(*
Nazwa:			P13_BottleTransfer
Opis:			Stacja odkładania butelek w różne miejsca
Wersja:			v0.1
Data:			2018-10-10
Autor:			DP
Urzadzenia:		
Konfiguracja:	
Info:

*)
PROGRAM P13_BottleTransfer
VAR_INPUT
	IbFirstFormCheckFormSensor				AT %I*	: BOOL; 						// Sygnal pierwszej formatki
	IbSecondFormCheckFormSensor				AT %I*	: BOOL; 						// Sygnal drugiej formatki
	IbBottleCheckAfterBottleTransferSensor	AT %I*	: BOOL; 						// Wejście z czujnika wykrycia butelki za robotem
	IbBottleTransferFormAfterSensor			AT %I*: BOOL; 					// Czujnik formatki za robotem
	IbBottleTransferFormAfterSensor2			AT %I*: BOOL; 					// Czujnik 2 formatki za robotem
END_VAR
VAR
	// Blok Sterujący podajnikiem nakrętek
	fbBottleTransfer									: FB_Robot2Bottles;
	tonEnableDelay: TON;
	eBottleTransferState					: E_Station;
	eBottleTransferRunningState				: E_RobotMovState;	
	fbBottleTransferState					: FB_State;	
	
	// WEJSCIA I WYJSCIA SPRZETOWE	
	QaDataRobotIO                            AT %Q*: ARRAY[1..8] OF USINT;
    QaDataRobotREG                           AT %Q*: ARRAY[1..32] OF UINT;
    IaDataRobotIO                            AT %I*: ARRAY[1..8] OF USINT;
    IaDataRobotREG                       	 AT %I*: ARRAY[1..32] OF UINT;
	

	
	
	TimerBottleTransferEnable: TOF;
	(*Nowe od robota Mitsubishi*)
	QbBottleTransferRobotMode1 AT %Q*:BOOL; 								//Zezwalanie na pracę robota 1
	QbBottleTransferRobotMode2 AT %Q*:BOOL; 								//Zezwalanie na pracę robota 2	

//	
	
	bBottleTransferLubricationResetCase: INT;
	tonBottleTransferLubricationResetCase1: TON;
	tonBottleTransferLubricationResetCase2: TON;
	tonBottleTransferLubricationResetCase3: TON;
	tonBottleTransferLubricationResetCase4: TON;
	tonBottleTransferLubricationResetCase5: TON;
	tonBottleTransferLubricationResetCase6: TON;
	tonBottleTransferLubricationResetCase7: TON;
	bTestWarning							: BOOL;
	bTestHoming								: BOOL;
	bTestPick								: BOOL;
	bTestPlace								: BOOL;
END_VAR

IF VIS.iBottleTransferPickOffsetZShow > 40	THEN
	VIS.iBottleTransferPickOffsetZShow								:= 40;
END_IF
IF VIS.iBottleTransferPickOffsetZShow < -60	THEN
	VIS.iBottleTransferPickOffsetZShow								:= -60;
END_IF

IF VIS.iBottleTransferPick2OffsetZShow > 40 THEN
	VIS.iBottleTransferPick2OffsetZShow								:= 40;
END_IF                                              				
IF VIS.iBottleTransferPick2OffsetZShow < -40 THEN   				
	VIS.iBottleTransferPick2OffsetZShow								:= -40;
END_IF                                              				
                                                    				
IF VIS.iBottleTransferPlace1OffsetZShow > 40 THEN   				
	VIS.iBottleTransferPlace1OffsetZShow							:= 40;
END_IF                                              				
IF VIS.iBottleTransferPlace1OffsetZShow < -60 THEN  				
	VIS.iBottleTransferPlace1OffsetZShow							:= -60;
END_IF

IF VIS.iBottleTransferPlace2OffsetZShow > 40 THEN
	VIS.iBottleTransferPlace2OffsetZShow							:= 40;
END_IF
IF VIS.iBottleTransferPlace2OffsetZShow < -80 THEN
	VIS.iBottleTransferPlace2OffsetZShow							:= -80;
END_IF

IF VIS.iBottleTransferPlace2OffsetXShow < -10 THEN
	VIS.iBottleTransferPlace2OffsetXShow							:= -10;
END_IF

IF VIS.iBottleTransferSpeedShow > 100 THEN
	VIS.iBottleTransferSpeedShow									:= 100;
END_IF
IF VIS.iBottleTransferSpeedShow < 5 THEN
	VIS.iBottleTransferSpeedShow									:= 5;
END_IF

aBottleTransfer();
aStatistics();
aManualMode();
(********* GENEROWANIE STANU STACJI DO WIZKI**********)		
fbBottleTransferState(
	eState															:= eBottleTransferState , 
	bRun															:= VIS.bBottleTransferRun,	
	eCapFeederRobotRunningState										:= eBottleTransferRunningState , 
	sStateDesc														=> VIS.sBottleTransferState,
	iState															=> VIS.iBottleTransferState	);	
(***** KONIEC GENEROWANIE STANU STACJI DO WIZKI*******)	

(*Opoznienie wyłączanie enabla*)
TimerBottleTransferEnable (IN:=bBottleTransferEnable , PT:=T#2S);

aWarning();


(**Wystawienie wyjść do robota**)

//QbBottleTransferRobotMode1											:= FALSE;
//QbBottleTransferRobotMode2											:= FALSE;

QbBottleTransferRobotMode1											:= TRUE;
QbBottleTransferRobotMode2											:= TRUE;

(**Koniec wystawienie wyjść do robota**)

ACTION aBottleTransfer:
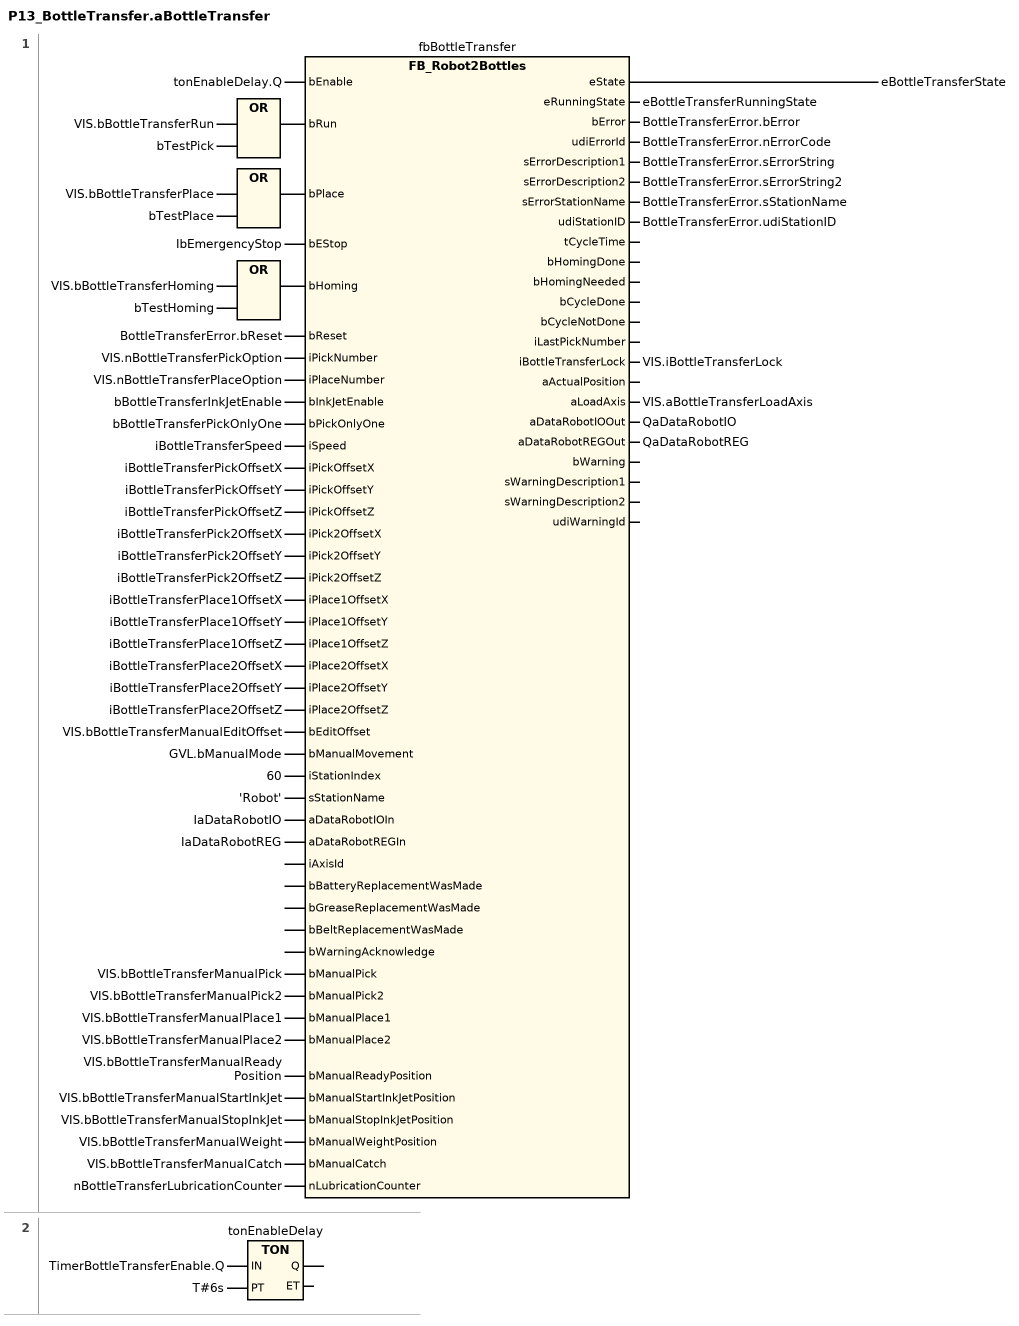
// NETWORK 1
fbBottleTransfer(
    bEnable := tonEnableDelay.Q,
    bRun := VIS.bBottleTransferRun OR bTestPick,
    bPlace := VIS.bBottleTransferPlace OR bTestPlace,
    bEStop := IbEmergencyStop,
    bHoming := VIS.bBottleTransferHoming OR bTestHoming,
    bReset := BottleTransferError.bReset,
    iPickNumber := VIS.nBottleTransferPickOption,
    iPlaceNumber := VIS.nBottleTransferPlaceOption,
    bInkJetEnable := bBottleTransferInkJetEnable,
    bPickOnlyOne := bBottleTransferPickOnlyOne,
    iSpeed := iBottleTransferSpeed,
    iPickOffsetX := iBottleTransferPickOffsetX,
    iPickOffsetY := iBottleTransferPickOffsetY,
    iPickOffsetZ := iBottleTransferPickOffsetZ,
    iPick2OffsetX := iBottleTransferPick2OffsetX,
    iPick2OffsetY := iBottleTransferPick2OffsetY,
    iPick2OffsetZ := iBottleTransferPick2OffsetZ,
    iPlace1OffsetX := iBottleTransferPlace1OffsetX,
    iPlace1OffsetY := iBottleTransferPlace1OffsetY,
    iPlace1OffsetZ := iBottleTransferPlace1OffsetZ,
    iPlace2OffsetX := iBottleTransferPlace2OffsetX,
    iPlace2OffsetY := iBottleTransferPlace2OffsetY,
    iPlace2OffsetZ := iBottleTransferPlace2OffsetZ,
    bEditOffset := VIS.bBottleTransferManualEditOffset,
    bManualMovement := GVL.bManualMode,
    iStationIndex := 60,
    sStationName := 'Robot',
    aDataRobotIOIn := IaDataRobotIO,
    aDataRobotREGIn := IaDataRobotREG,
    bManualPick := VIS.bBottleTransferManualPick,
    bManualPick2 := VIS.bBottleTransferManualPick2,
    bManualPlace1 := VIS.bBottleTransferManualPlace1,
    bManualPlace2 := VIS.bBottleTransferManualPlace2,
    bManualReadyPosition := VIS.bBottleTransferManualReadyPosition,
    bManualStartInkJetPosition := VIS.bBottleTransferManualStartInkJet,
    bManualStopInkJetPosition := VIS.bBottleTransferManualStopInkJet,
    bManualWeightPosition := VIS.bBottleTransferManualWeight,
    bManualCatch := VIS.bBottleTransferManualCatch,
    nLubricationCounter := nBottleTransferLubricationCounter,
    eRunningState => eBottleTransferRunningState,
    bError => BottleTransferError.bError,
    udiErrorId => BottleTransferError.nErrorCode,
    sErrorDescription1 => BottleTransferError.sErrorString,
    sErrorDescription2 => BottleTransferError.sErrorString2,
    sErrorStationName => BottleTransferError.sStationName,
    udiStationID => BottleTransferError.udiStationID,
    iBottleTransferLock => VIS.iBottleTransferLock,
    aLoadAxis => VIS.aBottleTransferLoadAxis,
    aDataRobotIOOut => QaDataRobotIO,
    aDataRobotREGOut => QaDataRobotREG); // FB_Robot2Bottles
eBottleTransferState := fbBottleTransfer.eState;

// NETWORK 2
tonEnableDelay(IN := TimerBottleTransferEnable.Q, PT := T#6s); // TON
END_ACTION

ACTION aManualMode:
	//iBottleTransferLock									:INT;					// Blokowanie przycisków trybu manualnego (b0-1 blokuj 
																					// 2#11111111 - nie moge nic  
																					// 2#11111110 - moge pobrać (tylko Pick1 i Pick 2 odblokowane)
																					// 2#11101001 - moge odłożyć, odrzucić i pojechać przed inkjet		
																					// 2#11110111 - moge jechać tylko do gotowości
																					// 2#11110111 - moge jechać tylko do gotowości
																					// 2#11011111 - moge jechać do koniec inkjet
																					// 2#10101101 - moge odłożyć na ety., wrocić przed inkjet
																					// 2#11111110 - moge pobrać
IF	 VIS.iBottleTransferLock = 2#11111111 THEN //2#11111111 - nie moge nic  
		VIS.bBottleTransferManualCatchVisibility				:= FALSE;					 	// Chwytak - przycisk odblokowany
  	  	VIS.bBottleTransferManualPickVisibility					:= FALSE; 						// Pobierz 1 but. - przycisk odblokowany
		VIS.bBottleTransferManualPick2Visibility 				:= FALSE; 						// Pobierz 2 but. - przycisk odblokowany
  	 	VIS.bBottleTransferManualPlace1Visibility				:= FALSE; 						// Odłóż na etykieciarkę - przycisk odblokowany
  	 	VIS.bBottleTransferManualPlace2Visibility				:= FALSE; 						// Odłóż na odrzut - przycisk odblokowany
  	 	VIS.bBottleTransferManualReadyPositionVisibility		:= FALSE; 						// Gotowość - przycisk odblokowany
		VIS.bBottleTransferManualStartInkJetVisibility			:= FALSE; 						// Start InkJet - przycisk odblokowany
		VIS.bBottleTransferManualStopInkJetVisibility			:= FALSE; 						// Stop InkJet - przycisk odblokowany	
ELSIF VIS.iBottleTransferLock = 2#11111110 THEN //2#11111110 - moge pobrać (tylko Pick1 i Pick 2 odblokowane)  
		VIS.bBottleTransferManualCatchVisibility				:= FALSE;					 	// Chwytak - przycisk odblokowany
  	  	VIS.bBottleTransferManualPickVisibility					:= TRUE; 						// Pobierz 1 but. - przycisk odblokowany
		VIS.bBottleTransferManualPick2Visibility 				:= TRUE;  						// Pobierz 2 but. - przycisk odblokowany
  	 	VIS.bBottleTransferManualPlace1Visibility				:= FALSE; 						// Odłóż na etykieciarkę - przycisk odblokowany
  	 	VIS.bBottleTransferManualPlace2Visibility				:= FALSE; 						// Odłóż na odrzut - przycisk odblokowany
  	 	VIS.bBottleTransferManualReadyPositionVisibility		:= FALSE; 						// Gotowość - przycisk odblokowany
		VIS.bBottleTransferManualStartInkJetVisibility			:= FALSE; 						// Start InkJet - przycisk odblokowany
		VIS.bBottleTransferManualStopInkJetVisibility			:= FALSE; 						// Stop InkJet - przycisk odblokowany		
ELSIF VIS.iBottleTransferLock = 2#11101001 THEN //2#11101001 - moge odłożyć, odrzucić i pojechać przed inkjet	
 		VIS.bBottleTransferManualCatchVisibility				:= FALSE;					 	// Chwytak - przycisk odblokowany
  	  	VIS.bBottleTransferManualPickVisibility					:= FALSE; 						// Pobierz 1 but. - przycisk odblokowany
		VIS.bBottleTransferManualPick2Visibility 				:= FALSE; 						// Pobierz 2 but. - przycisk odblokowany
  	 	VIS.bBottleTransferManualPlace1Visibility				:= TRUE; 						// Odłóż na etykieciarkę - przycisk odblokowany
  	 	VIS.bBottleTransferManualPlace2Visibility				:= TRUE;  						// Odłóż na odrzut - przycisk odblokowany
  	 	VIS.bBottleTransferManualReadyPositionVisibility		:= FALSE; 						// Gotowość - przycisk odblokowany
		VIS.bBottleTransferManualStartInkJetVisibility			:= TRUE;  						// Start InkJet - przycisk odblokowany
		VIS.bBottleTransferManualStopInkJetVisibility			:= FALSE; 						// Stop InkJet - przycisk odblokowany	
ELSIF VIS.iBottleTransferLock = 2#11110111 THEN //2#11110111 - moge jechać tylko do gotowości 
		VIS.bBottleTransferManualCatchVisibility				:= FALSE;					 	// Chwytak - przycisk odblokowany
  	  	VIS.bBottleTransferManualPickVisibility					:= FALSE; 						// Pobierz 1 but. - przycisk odblokowany
		VIS.bBottleTransferManualPick2Visibility 				:= FALSE; 						// Pobierz 2 but. - przycisk odblokowany
  	 	VIS.bBottleTransferManualPlace1Visibility				:= FALSE; 						// Odłóż na etykieciarkę - przycisk odblokowany
  	 	VIS.bBottleTransferManualPlace2Visibility				:= FALSE; 						// Odłóż na odrzut - przycisk odblokowany
  	 	VIS.bBottleTransferManualReadyPositionVisibility		:= TRUE; 						// Gotowość - przycisk odblokowany
		VIS.bBottleTransferManualStartInkJetVisibility			:= FALSE; 						// Start InkJet - przycisk odblokowany
		VIS.bBottleTransferManualStopInkJetVisibility			:= FALSE; 						// Stop InkJet - przycisk odblokowany	
ELSIF VIS.iBottleTransferLock = 2#11110111 THEN //2#11110111 - moge jechać tylko do gotowości 
		VIS.bBottleTransferManualCatchVisibility				:= FALSE;					 	// Chwytak - przycisk odblokowany
  	  	VIS.bBottleTransferManualPickVisibility					:= FALSE; 						// Pobierz 1 but. - przycisk odblokowany
		VIS.bBottleTransferManualPick2Visibility 				:= FALSE; 						// Pobierz 2 but. - przycisk odblokowany
  	 	VIS.bBottleTransferManualPlace1Visibility				:= FALSE; 						// Odłóż na etykieciarkę - przycisk odblokowany
  	 	VIS.bBottleTransferManualPlace2Visibility				:= FALSE; 						// Odłóż na odrzut - przycisk odblokowany
  	 	VIS.bBottleTransferManualReadyPositionVisibility		:= TRUE;  						// Gotowość - przycisk odblokowany
		VIS.bBottleTransferManualStartInkJetVisibility			:= FALSE; 						// Start InkJet - przycisk odblokowany
		VIS.bBottleTransferManualStopInkJetVisibility			:= FALSE; 						// Stop InkJet - przycisk odblokowany	
ELSIF VIS.iBottleTransferLock = 2#11011111 THEN //2#11011111 - moge jechać do koniec inkjet  
		VIS.bBottleTransferManualCatchVisibility				:= FALSE;					 	// Chwytak - przycisk odblokowany
  	  	VIS.bBottleTransferManualPickVisibility					:= FALSE; 						// Pobierz 1 but. - przycisk odblokowany
		VIS.bBottleTransferManualPick2Visibility 				:= FALSE; 						// Pobierz 2 but. - przycisk odblokowany
  	 	VIS.bBottleTransferManualPlace1Visibility				:= FALSE; 						// Odłóż na etykieciarkę - przycisk odblokowany
  	 	VIS.bBottleTransferManualPlace2Visibility				:= FALSE; 						// Odłóż na odrzut - przycisk odblokowany
  	 	VIS.bBottleTransferManualReadyPositionVisibility		:= FALSE; 						// Gotowość - przycisk odblokowany
		VIS.bBottleTransferManualStartInkJetVisibility			:= FALSE; 						// Start InkJet - przycisk odblokowany
		VIS.bBottleTransferManualStopInkJetVisibility			:= TRUE;  						// Stop InkJet - przycisk odblokowany	
ELSIF VIS.iBottleTransferLock = 2#10101101 THEN //2#10101101 - moge odłożyć na ety., wrocić przed inkjet  
		VIS.bBottleTransferManualCatchVisibility				:= FALSE;					 	// Chwytak - przycisk odblokowany
  	  	VIS.bBottleTransferManualPickVisibility					:= FALSE; 						// Pobierz 1 but. - przycisk odblokowany
		VIS.bBottleTransferManualPick2Visibility 				:= FALSE; 						// Pobierz 2 but. - przycisk odblokowany
  	 	VIS.bBottleTransferManualPlace1Visibility				:= TRUE;  						// Odłóż na etykieciarkę - przycisk odblokowany
  	 	VIS.bBottleTransferManualPlace2Visibility				:= FALSE; 						// Odłóż na odrzut - przycisk odblokowany
  	 	VIS.bBottleTransferManualReadyPositionVisibility		:= FALSE; 						// Gotowość - przycisk odblokowany
		VIS.bBottleTransferManualStartInkJetVisibility			:= TRUE;  						// Start InkJet - przycisk odblokowany
		VIS.bBottleTransferManualStopInkJetVisibility			:= FALSE; 						// Stop InkJet - przycisk odblokowany	
ELSIF VIS.iBottleTransferLock = 2#11111110 THEN //2#11111110 - moge pobrać 	
		VIS.bBottleTransferManualCatchVisibility				:= FALSE;					 	// Chwytak - przycisk odblokowany
  	  	VIS.bBottleTransferManualPickVisibility					:= TRUE;						// Pobierz 1 but. - przycisk odblokowany
		VIS.bBottleTransferManualPick2Visibility 				:= FALSE; 						// Pobierz 2 but. - przycisk odblokowany
  	 	VIS.bBottleTransferManualPlace1Visibility				:= FALSE; 						// Odłóż na etykieciarkę - przycisk odblokowany
  	 	VIS.bBottleTransferManualPlace2Visibility				:= FALSE; 						// Odłóż na odrzut - przycisk odblokowany
  	 	VIS.bBottleTransferManualReadyPositionVisibility		:= FALSE; 						// Gotowość - przycisk odblokowany
		VIS.bBottleTransferManualStartInkJetVisibility			:= FALSE; 						// Start InkJet - przycisk odblokowany
		VIS.bBottleTransferManualStopInkJetVisibility			:= FALSE; 						// Stop InkJet - przycisk odblokowany	
END_IF
END_ACTION

ACTION aStatistics:
VIS.iBottleTransferState				;
VIS.sBottleTransferState				;
VIS.bBottleTransferHoming				;
VIS.bBottleTransferHeightSet 			;
VIS.bBottleTransferIgnoreErrors			;
VIS.bBottleTransferRun					;
VIS.bBottleTransferPlace				;
VIS.nBottleTransferPlaceOption			;
VIS.nBottleTransferPickOption			;
VIS.bBottleTransferManualCatch			;
VIS.bBottleTransferManualPick			;
VIS.bBottleTransferManualPick2 			;
VIS.bBottleTransferManualPlace1			;
VIS.bBottleTransferManualPlace2			;
VIS.bBottleTransferManualReadyPosition	;
VIS.bBottleTransferManualStartInkJet	;
VIS.bBottleTransferManualStopInkJet		;
VIS.bBottleTransferManualEditOffset		;
VIS.bBottleTransferAllFormsToLabeler	;
VIS.bBottleTransferAllFormsToExit		;
VIS.bBottleTransferLubricationReset		;
VIS.aBottleTransferLoadAxis				;
VIS.iBottleTransferLock					;
END_ACTION

ACTION aWarning:
(****Ostrzezenia***)

//BottleTransferWarning[1].sDescription								:= 'Przeprowadzić smarowanie i przegląd techniczny robota';
BottleTransferWarning[1].sDescription								:= fbBottleTransfer.sWarningDescription1;
IF BottleTransferWarning[1].sDescription = '' THEN
	BottleTransferWarning[1].sDescription := 'Robot | Ostrzeżenie';
END_IF
//IF nBottleTransferLubricationCounter>900000 AND NOT BottleTransferWarning[1].bWarning THEN

tonBottleTransferLubricationResetCase1 	(IN:=bBottleTransferLubricationResetCase=10 OR bBottleTransferLubricationResetCase=300, PT:=T#1S);
tonBottleTransferLubricationResetCase2 	(IN:=bBottleTransferLubricationResetCase=100 OR bBottleTransferLubricationResetCase=200, PT:=T#1S);
tonBottleTransferLubricationResetCase3 	(IN:=bBottleTransferLubricationResetCase=110 OR bBottleTransferLubricationResetCase=210, PT:=T#1S);
tonBottleTransferLubricationResetCase4 	(IN:=bBottleTransferLubricationResetCase=120 OR bBottleTransferLubricationResetCase=220, PT:=T#1S);
tonBottleTransferLubricationResetCase5 	(IN:=bBottleTransferLubricationResetCase=130 OR bBottleTransferLubricationResetCase=230, PT:=T#1S);
tonBottleTransferLubricationResetCase6 	(IN:=bBottleTransferLubricationResetCase=140 OR bBottleTransferLubricationResetCase=240, PT:=T#1S);
tonBottleTransferLubricationResetCase7 	(IN:=bBottleTransferLubricationResetCase=150 OR bBottleTransferLubricationResetCase=250, PT:=T#1S);

IF (fbBottleTransfer.bWarning OR bTestWarning) AND NOT BottleTransferWarning[1].bWarning THEN
	BottleTransferWarning[1].bWarning								:= TRUE;
	BottleTransferWarning[1].udiWarningCode							:= 58;
ELSIF BottleTransferWarning[1].bAcknowledge THEN
	
	CASE bBottleTransferLubricationResetCase OF 
		
		0:
			fbBottleTransfer.iAxisId					:= 0 ;
			fbBottleTransfer.bBatteryReplacementWasMade	:= FALSE;			
			fbBottleTransfer.bGreaseReplacementWasMade	:= FALSE;		
			fbBottleTransfer.bBeltReplacementWasMade	:= FALSE;		
			fbBottleTransfer.bWarningAcknowledge		:= FALSE;		

			//battery
			//1330,0111,7450,7451,7510,7520			
			//grease
			//7121,7122,7123,7124,7125,7126,7530			
			//belt
			//7131,7132,7133,7134,7135,7136,7540
			
			IF	//baterry 
				fbBottleTransfer.udiWarningId =	1330 OR fbBottleTransfer.udiWarningId =	0111 OR	
				fbBottleTransfer.udiWarningId =	7450 OR fbBottleTransfer.udiWarningId =	7451 OR
				fbBottleTransfer.udiWarningId =	7510 OR fbBottleTransfer.udiWarningId =	7520 		
				THEN
				bBottleTransferLubricationResetCase	:=	10;
			ELSIF	//grease
				fbBottleTransfer.udiWarningId =	7121 OR fbBottleTransfer.udiWarningId =	7122 OR	
				fbBottleTransfer.udiWarningId =	7123 OR fbBottleTransfer.udiWarningId =	7124 OR
				fbBottleTransfer.udiWarningId =	7125 OR fbBottleTransfer.udiWarningId =	7126 OR
				fbBottleTransfer.udiWarningId =	7530 
				THEN
				bBottleTransferLubricationResetCase	:=	100;
			ELSIF	//belt
				fbBottleTransfer.udiWarningId =	7131 OR fbBottleTransfer.udiWarningId =	7132 OR	
				fbBottleTransfer.udiWarningId =	7133 OR fbBottleTransfer.udiWarningId =	7134 OR
				fbBottleTransfer.udiWarningId =	7135 OR fbBottleTransfer.udiWarningId =	7136 OR
				fbBottleTransfer.udiWarningId =	7540 
				THEN
				bBottleTransferLubricationResetCase	:=	200;
			ELSE	//other
				bBottleTransferLubricationResetCase	:=	300;
						
			END_IF
			
		10: //battery
			fbBottleTransfer.bBatteryReplacementWasMade	:=	TRUE;			
			fbBottleTransfer.bWarningAcknowledge		:=	TRUE;
			IF tonBottleTransferLubricationResetCase1.Q THEN
				bBottleTransferLubricationResetCase		:=	1000;
			END_IF
		
		100: //grease
			fbBottleTransfer.iAxisId					:= 1 ;	
			fbBottleTransfer.bGreaseReplacementWasMade	:= TRUE;		
			fbBottleTransfer.bWarningAcknowledge		:= TRUE;
			IF tonBottleTransferLubricationResetCase2.Q THEN
				bBottleTransferLubricationResetCase		:=	bBottleTransferLubricationResetCase	+	10;
			END_IF
		110://grease
			fbBottleTransfer.iAxisId					:= 2 ;	
			fbBottleTransfer.bGreaseReplacementWasMade	:= TRUE;		
			fbBottleTransfer.bWarningAcknowledge		:= TRUE;
			IF tonBottleTransferLubricationResetCase3.Q THEN
				bBottleTransferLubricationResetCase		:=	bBottleTransferLubricationResetCase	+	10;
			END_IF			
		120: //grease
			fbBottleTransfer.iAxisId					:= 3 ;	
			fbBottleTransfer.bGreaseReplacementWasMade	:= TRUE;		
			fbBottleTransfer.bWarningAcknowledge		:= TRUE;
			IF tonBottleTransferLubricationResetCase4.Q THEN
				bBottleTransferLubricationResetCase		:=	bBottleTransferLubricationResetCase	+	10;
			END_IF	
		130://grease
			fbBottleTransfer.iAxisId					:= 4 ;	
			fbBottleTransfer.bGreaseReplacementWasMade	:= TRUE;		
			fbBottleTransfer.bWarningAcknowledge		:= TRUE;
			IF tonBottleTransferLubricationResetCase5.Q THEN
				bBottleTransferLubricationResetCase		:=	bBottleTransferLubricationResetCase	+	10;
			END_IF	
		140://grease
			fbBottleTransfer.iAxisId					:= 5 ;	
			fbBottleTransfer.bGreaseReplacementWasMade	:= TRUE;		
			fbBottleTransfer.bWarningAcknowledge		:= TRUE;
			IF tonBottleTransferLubricationResetCase6.Q THEN
				bBottleTransferLubricationResetCase		:=	bBottleTransferLubricationResetCase	+	10;
			END_IF	
		150://grease
			fbBottleTransfer.iAxisId					:= 6 ;	
			fbBottleTransfer.bGreaseReplacementWasMade	:= TRUE;		
			fbBottleTransfer.bWarningAcknowledge		:= TRUE;
			IF tonBottleTransferLubricationResetCase7.Q THEN
				bBottleTransferLubricationResetCase		:=	1000;;
			END_IF				
			
		200: //belt
			fbBottleTransfer.iAxisId					:= 1 ;	
			fbBottleTransfer.bBeltReplacementWasMade	:= TRUE;		
			fbBottleTransfer.bWarningAcknowledge		:= TRUE;		
			IF tonBottleTransferLubricationResetCase2.Q  THEN
				bBottleTransferLubricationResetCase		:=	bBottleTransferLubricationResetCase	+	10;
			END_IF
		210: //belt
			fbBottleTransfer.iAxisId					:= 2 ;	
			fbBottleTransfer.bBeltReplacementWasMade	:= TRUE;		
			fbBottleTransfer.bWarningAcknowledge		:= TRUE;		
			IF tonBottleTransferLubricationResetCase3.Q THEN
				bBottleTransferLubricationResetCase		:=	bBottleTransferLubricationResetCase	+	10;
			END_IF		
		220: //belt
			fbBottleTransfer.iAxisId					:= 3 ;	
			fbBottleTransfer.bBeltReplacementWasMade	:= TRUE;		
			fbBottleTransfer.bWarningAcknowledge		:= TRUE;		
			IF (*tonBottleTransferLubricationResetCase4.Q*) fbBottleTransfer.bBeltReplenishmentFinished THEN
				bBottleTransferLubricationResetCase		:=	bBottleTransferLubricationResetCase	+	10;
			END_IF	
		230: //belt
			fbBottleTransfer.iAxisId					:= 4 ;	
			fbBottleTransfer.bBeltReplacementWasMade	:= TRUE;		
			fbBottleTransfer.bWarningAcknowledge		:= TRUE;		
			IF (*tonBottleTransferLubricationResetCase5.Q*) fbBottleTransfer.bBeltReplenishmentFinished THEN
				bBottleTransferLubricationResetCase		:=	bBottleTransferLubricationResetCase	+	10;
			END_IF	
		240: //belt
			fbBottleTransfer.iAxisId					:= 5;	
			fbBottleTransfer.bBeltReplacementWasMade	:= TRUE;		
			fbBottleTransfer.bWarningAcknowledge		:= TRUE;		
			IF tonBottleTransferLubricationResetCase6.Q THEN
				bBottleTransferLubricationResetCase		:=	bBottleTransferLubricationResetCase	+	10;
			END_IF	
		250: //belt
			fbBottleTransfer.iAxisId					:= 6 ;	
			fbBottleTransfer.bBeltReplacementWasMade	:= TRUE;		
			fbBottleTransfer.bWarningAcknowledge		:= TRUE;		
			IF tonBottleTransferLubricationResetCase7.Q THEN
				bBottleTransferLubricationResetCase		:=	1000;
			END_IF	
			
		300://Other		
			fbBottleTransfer.bWarningAcknowledge		:=	TRUE;
			IF tonBottleTransferLubricationResetCase1.Q THEN
				bBottleTransferLubricationResetCase		:=	1000;
			END_IF
		
		1000: //end
		
			fbBottleTransfer.iAxisId					:= 0 ;
			fbBottleTransfer.bBatteryReplacementWasMade	:= FALSE;			
			fbBottleTransfer.bGreaseReplacementWasMade	:= FALSE;		
			fbBottleTransfer.bBeltReplacementWasMade	:= FALSE;		
			fbBottleTransfer.bWarningAcknowledge		:= FALSE;	
		
			bBottleTransferLubricationResetCase								:= 0;
			BottleTransferWarning[1].bWarning								:= FALSE;
			BottleTransferWarning[1].bAcknowledge							:= FALSE;
			VIS.uliWarningAcknowledge.5 										:= FALSE;
			//nBottleTransferLubricationCounter 								:= 0;
			VIS.bBottleTransferLubricationReset 							:= FALSE;
	
	END_CASE
	


	
END_IF
END_ACTION

END_PROGRAM

(* stored: Version 1.1.0.1, ProductVersion 3.1.4026.13, FileIdentifier b0585e14b99c238be491003b598066f728fb4736, FileSignature 7c5812ce284e299d043454f3df4f0bd3c0c5d9cd99988f692b754fe152e028ddd4b0e0b78d3d1c7259bf52354ba6449ef88bc349303d6b8f3f40f6c979c4dc11f8da61d6d7306bb3adea25ead6a1cec0171e410a2c59c00b0877065574425a1cff1a512acc5cdcc400ab8bcb3c103994cd1890f23b52f28e399f296a8dd8b37864947cd59d3f46c7f7648c9a6487d7fed36b0771e26f644396245d9c93311821864574ac25fb4f1713178561ea1de65dc5f4e697faef98c6e95c04b0581a1b3bde307aa38ebf425e6a4381d7a3b688c96243a0280903f2765997041d8e5ffd956fe5443e12bd434461200d15cdc5e87e715c3099be7461f171f48bc0fc30a2ce
   POU P13_BottleTransfer: Id {448f8d44-051a-4fc5-a96f-f0891c98611d}, SpecialFunc None
   Action aBottleTransfer: Id {dbb67d15-01a9-4455-97b3-b17140757e83}
   Action aManualMode: Id {d4d46939-cdba-4d81-82c9-62667809ed20}
   Action aStatistics: Id {8a8dfdb6-de92-4a1c-b258-094691bdf502}
   Action aWarning: Id {f520abdd-237d-4b26-9d09-8107af858b13} *)
